KUKA KRL data list: vw_usr_r.dat

&ACCESS RV1
&REL 1
&PARAM TPVW_VERSION = 3.3.5
DEFDAT  VW_USR_R
; FOLD ;%{H}%MKUKATPVW
; ENDFOLD
ENDDAT
